% RSLogix 500 project WATER_TANK_CONTROL_BAK000.RSS, saved by version 8.30.00.16 %
PROJECT "1761-L16"    % processor: Bul.1763 MicroLogix 1100 Series B %

PROGRAM FILES
  LAD 2   6 rungs

DATA FILES
  O0 OUTPUT  4 elements
  I1 INPUT  6 elements
  S2 STATUS  66 elements
  B3 BINARY  1 elements
  T4 TIMER  1 elements
  C5 COUNTER  1 elements
  R6 CONTROL  1 elements
  N7 INTEGER  1 elements
  F8 FLOAT  1 elements

LADDER 2
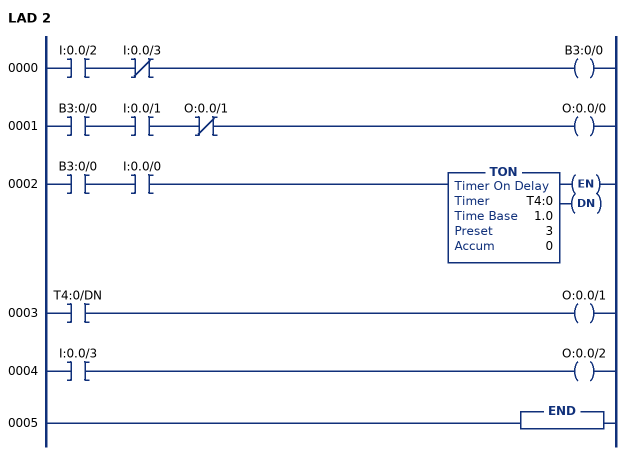
% Rung: 0 %  % edit flag set %
SOR XIC I:0.0/2 XIO I:0.0/3 OTE B3:0/0 EOR
% Rung: 1 %  % edit flag set %
SOR XIC B3:0/0 XIC I:0.0/1 XIO O:0.0/1 OTE O:0.0/0 EOR
% Rung: 2 %  % edit flag set %
SOR XIC B3:0/0 XIC I:0.0/0 TON T4:0 1.0 3 0 EOR
% Rung: 3 %  % edit flag set %
SOR XIC T4:0/DN OTE O:0.0/1 EOR
% Rung: 4 %  % edit flag set %
SOR XIC I:0.0/3 OTE O:0.0/2 EOR
% Rung: 5 %
SOR END EOR
